// TIA Portal V19 export
DATA_BLOCK "Gestion_DB"   // DB5
// stored: InstanceOfName Gestion, InstanceOfType FB
"Gestion"
   // VAR RETAIN
   //    "Code erreur" : Word;
   //    "FM Noires" : Bool;
   //    "FM Mauvaises" : Bool;
   //    "FM Bonnes" : Bool;
   //    "FM QuiSertARien" : Bool;
   // END_VAR
BEGIN
END_DATA_BLOCK
